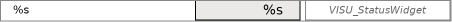
VISUALIZATION VISU_Measurement  // 452x22
VAR_IN_OUT
    widget : MeasurementWidget;
END_VAR
    Rectangle (10,0 180x20), "%s", text variable: widget.name
    Rectangle (195,0 105x20)
    Frame (305,0 145x20)
        shows VISU_StatusWidget(widget := widget.actualStatusWidget)
    Rectangle (195,0 100x20), "%s", text variable: widget.display
END_VISUALIZATION

(* stored: Version 1.1.0.1, ProductVersion 3.1.4019.2
   Visu VISU_Measurement: Id {13c95a8a-de6b-42c2-9ac7-73ccca01f0b2} *)
